PROGRAM PRG_Roughing_Control
VAR
	
END_VAR

END_PROGRAM

(* stored: Version 1.1.0.1, ProductVersion 3.1.4022.18
   POU PRG_Roughing_Control: Id {87120f5c-8975-4cdd-a125-ee85e558c6d5}, SpecialFunc None *)
